ABB RobotStudio station: RobotStudioDemo.rsstn

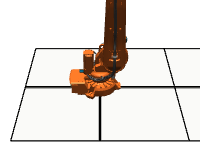
Station RobotStudioDemo (saved by RobotStudio 6.7.7985.1011)
Controller IRB_4600_40kg_2.55m
  mechanical unit ROB_1: IRB4600_40_255__02, 6 joints, base frame (0, 0, 0) mm
Layout (positions relative to the parent item):
  - IRB4600_40_255__02 [mechanism, from Robots\IRB4600_40_255__02.rslib] at (0, 0, 0) mm; joint values [0, 0, 0, 0, 0.5236, 0] (rad or m)
